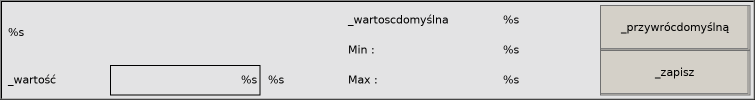
VISUALIZATION F_Descriptor  // 755x100
VAR_IN_OUT
	stData 	: ST_BaseHMIDescriptorEdit;
END_VAR
    Rectangle (0,0 755x100)
    Rectangle (5,5 330x55), "%s", text variable: stData.wsText
    Rectangle (345,35 100x30), "Min :"
    Rectangle (345,65 100x30), "Max :"
    Rectangle (345,5 150x30), "_wartoscdomyślna", text list: 'TextList_02', text index: 1
    Rectangle (500,5 50x30), "%s", text variable: stData.rDefaultValue, text list: 'TextList_02', text index: 1
    Rectangle (500,35 50x30), "%s", text variable: stData.rMin
    Rectangle (500,65 50x30), "%s", text variable: stData.rMax
    Rectangle (5,65 100x30), "_wartość"
    Rectangle (110,65 150x30), "%s", text variable: stData.rValue
        OnMouseDown: write the text variable via KlawiaturaCyfry, min stData.rMin, max stData.rMax
    Rectangle (265,65 70x30), "%s", text variable: stData.sUnit
    Button (600,5 150x45), "_przywrócdomyślną", text list: 'TextList_02', text index: 3
        OnMouseDown: execute { stData.bSetDefault := TRUE; }
    Button (600,50 150x45), "_zapisz", text list: 'TextList_02', text index: 4
        OnMouseDown: execute { stData.bSave := TRUE; }
END_VISUALIZATION

(* stored: Version 1.1.0.1
   Visu F_Descriptor: Id {0d1b9a85-585f-06b8-2f22-51c48921c009} *)
